(* CODESYS project zadanie_z_zajęć.project

Project tree, tasks and I/O mapping:
  Device : CODESYS Control Win V3, CODESYS, version 3.5.20.30
    application Application
      libraries: Standard, 3.5.18.0 (System)
      task VISU_TASK (cyclic, interval 100 ms, priority 31) calls VisuElems.Visu_Prg
      task MainTask (cyclic, interval t#20ms, priority 1) calls PLC_PRG_GK
      visualisation Visualization
      program PLC_PRG_GK [LD]
  libraries: Standard, 3.5.18.0 (System); VisuElemBase, * (System)
  text list GlobalTextList
*)

// Device/Application/PLC_PRG_GK
PROGRAM PLC_PRG_GK
VAR
    S1_GK, S2_GK:BOOL;
	S2_SET_GK:BOOL;
	
    S1_mono_GK, S1_bi_GK, S2_mono_GK, S2_bi_GK, S3_mono_GK, S3_bi_GK: BOOL;
    H1_GK, H2_GK, H3_GK: BOOL;
    H4_GK, H5_GK, H6_GK: BOOL;
 	M1_GK, M2_GK, M3_GK: BOOL;
    M4_GK, M5_GK, M6_GK: BOOL;
	S2_nacisniecia_GK: WORD :=3;
	S1_impuls_GK: TIME := T#5S;
	S2_impuls_GK: TIME := T#3S;
	S2_2_impuls_GK: TIME := T#6S;
	
	reset_GK:BOOL;
	S3_GK: BOOL;
	TP_GK: TP;
	
	TP2_GK: TP;
	F_TRIG_GK: F_TRIG;
	TOF_GK: TOF;
	TP3_GK: TP;
	TON_GK: TON;
	TON2_GK: TON;
	TON3_GK: TON;
END_VAR
VAR // added by the converter: edge detectors and wires of the graphical bodies
    _w1, _w2 : BOOL;
END_VAR

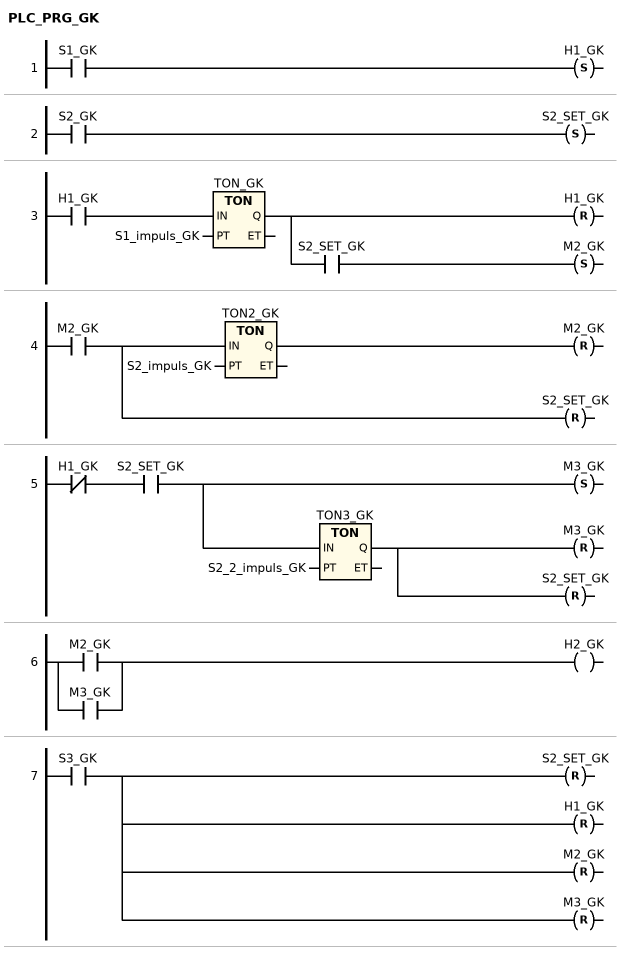
// NETWORK 1
H1_GK S= S1_GK;

// NETWORK 2
S2_SET_GK S= S2_GK;

// NETWORK 3
TON_GK(IN := H1_GK, PT := S1_impuls_GK); // TON
H1_GK R= TON_GK.Q;
M2_GK S= TON_GK.Q AND S2_SET_GK;

// NETWORK 4
_w1 := M2_GK;
TON2_GK(IN := _w1, PT := S2_impuls_GK); // TON
M2_GK R= TON2_GK.Q;
S2_SET_GK R= _w1;

// NETWORK 5
_w2 := NOT H1_GK AND S2_SET_GK;
M3_GK S= _w2;
TON3_GK(IN := _w2, PT := S2_2_impuls_GK); // TON
M3_GK R= TON3_GK.Q;
S2_SET_GK R= TON3_GK.Q;

// NETWORK 6
H2_GK := M2_GK OR M3_GK;

// NETWORK 7
S2_SET_GK R= S3_GK;
H1_GK R= S3_GK;
M2_GK R= S3_GK;
M3_GK R= S3_GK;

END_PROGRAM

// Device/Application/Visualization
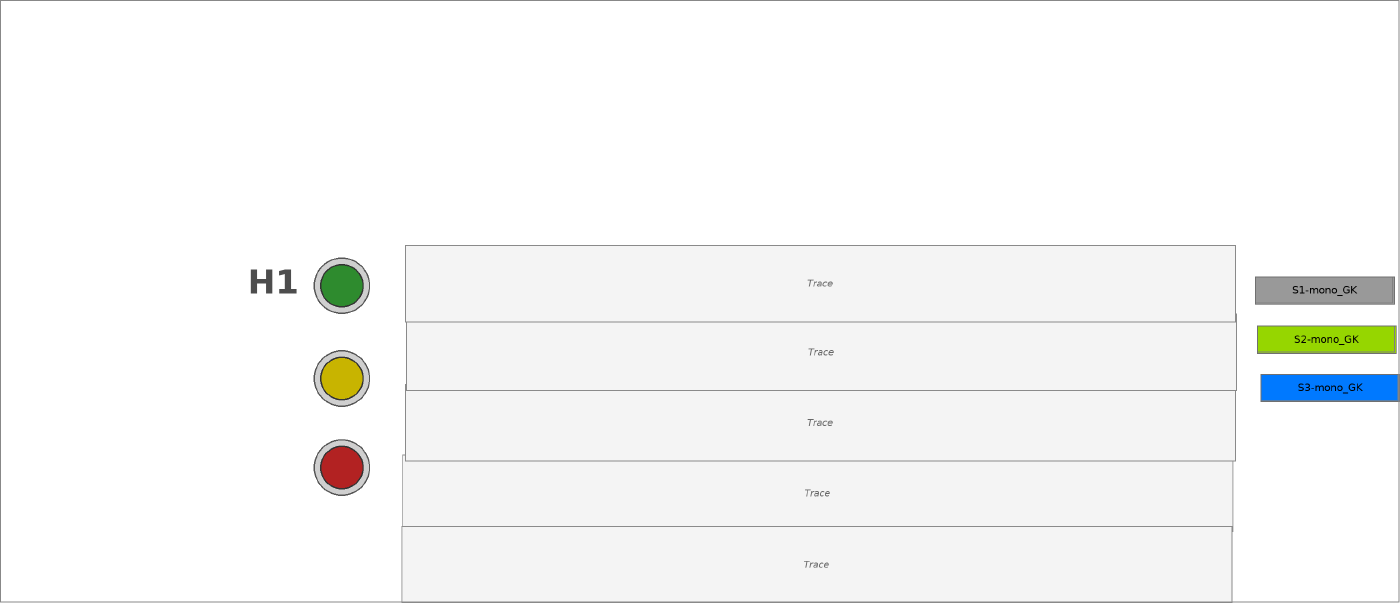
VISUALIZATION Visualization  // 1507x650
    Lamp1 (333,273 70x70), variable: PLC_PRG_GK.H1_GK, style: Lamp-Lamp1-Green
    Lamp1 (333,373 70x70), variable: PLC_PRG_GK.H2_GK, style: Lamp-Lamp1-Yellow
    Lamp1 (333,469 70x70), variable: PLC_PRG_GK.H3_GK, style: Lamp-Lamp1-Red
    Button (1351,298 150x30), "S1-mono_GK"
        tap PLC_PRG_GK.S1_GK
    Button (1353,351 150x30), "S2-mono_GK"
        tap PLC_PRG_GK.S2_GK
    Button (1357,403 150x30), "S3-mono_GK"
        tap PLC_PRG_GK.S3_GK
    Label (219,289 150x30), "H1"
    Trace (433,490 894x83)
    Trace (436,414 894x83)
    Trace (437,338 894x83)
    Trace (436,264 894x83)
    Trace (432,567 894x83)
END_VISUALIZATION
